// TIA Portal V17 export
// export: Created 2025-03-05T08:03:48.3158656Z, ExportSetting WithDefaults, DisplayName Totally Integrated Automation Portal, DisplayVersion V17 Update 8, DisplayName TIA Portal Openness, DisplayVersion V17 Update 8, DisplayName TIA Portal Version Control Interface, DisplayVersion V17, DisplayName SINAMICS Startdrive Advanced, DisplayVersion V17 SP2, DisplayName SINAMICS Startdrive G110M, G120, G120C, G120D, G120P, G115D, DisplayVersion V17 SP2, DisplayName SINAMICS Startdrive G130, G150, S120, S150, SINAMICS MV, S210, DisplayVersion V17 SP2, DisplayName STEP 7 Professional, DisplayVersion V17 Update 8, DisplayName SINUMERIK ONE STEP 7 Toolbox, DisplayVersion V17 Update 12, DisplayName SINUMERIK 840D sl STEP 7 Toolbox, DisplayVersion V17 Update 12, DisplayName STEP 7 Safety, DisplayVersion V17 Update 6, DisplayName WinCC Advanced, DisplayVersion V17 Update 8
TYPE "HOPPER"
// stored: IsFailsafeCompliant false
   STRUCT
      PRESSURIZE_PROP_GAS_VALVE_F : Int;   // PRESSURIZE PROPORTIONAL GAS VALVE FEEDBACK
      PRESSURIZE_GAS_VALVE : Bool;   // HOPPER PRESSURIZE GAS VALVE STATUS (CLOSED = 0 / OPEN = 1)
      RELIEF_GAS_VALVE : Bool;   // HOPPER RELIEF GAS VALVE STATUS (CLOSED = 0 / OPEN = 1)
      HIGH_LEVEL : Bool;   // HOPPER HIGH LEVEL SENSOR STATUS (LEVEL NOT REACHED = 0 / LEVEL REACHED= 1)
      LOW_LEVEL : Bool;   // HOPPER LOW LEVEL SENSOR STATUS (LEVEL NOT REACHED = 0 / LEVEL REACHED= 1)
      MAX_WEIGHT_SETPOINT : Real;   // MAX WEIGHT SETPOINT (kg)
      TOTAL_WEIGHT : Real;   // TOTAL WEIGHT (kg)
      HOPPER_WEIGHT_SETPOINT : Real;   // HOPPER HMI SET WEIGHT (kg)
      POWDER_WEIGHT : Real;   // POWDER WEIGHT (kg)
      UPPER_JACKET_TEMPERATURE : Real;   // HOPPER UPPER JACKET TEMPERATURE VALUE (ºC)
      UPPER_JACKET_TEMPERATURE_SETPOINT : Real;   // HOPPER UPPER JACKET TEMPERATURE SETPOINT VALUE (ºC)
      LOWER_JACKET_TEMPERATURE : Real;   // HOPPER LOWER JACKET TEMPERATURE VALUE (ºC)
      LOWER_JACKET_TEMPERATURE_SETPOINT : Real;   // HOPPER LOWER JACKET TEMPERATURE SETPOINT VALUE (ºC)
      HOPPER_PRESSURE : Real;   // HOPPER COVER PRESSURE VALUE (Bar)
      HOPPER_PRESSURE_SETPOINT : Real;   // HOPPER COVER PRESSURE SETPOINT VALUE (Bar)
      STIRRER_CURRENT : DInt;   // HOPPER STIRRER CURRENT VALUE (mA)
      STIRRER_SPEED : DInt;   // HOPPER STIRRER SPEED VALUE (RPM or %)
      STIRRER_SPEED_SETPOINT : DInt;   // HOPPER STIRRER SPEED SETPOINT VALUE (RPM or %)
      TRANSFER_POWDER_VALVE : Bool;   // HOPPER TRANSFER POWDER VALVE STATUS (CLOSED = 0 / OPEN = 1)
      CLEANING_AIR_VALVE : Bool;
      LOAD_FEEDER_SEQ : Bool;
      POWDER_FLOW : Array[1..20] of "MEDICOAT_TIME_STAMP";   // HOPPER POWDER FLOW VALUE (Raw)
   END_STRUCT;
END_TYPE
